// TIA Portal V20 export
DATA_BLOCK "DB_BadPartOnFixture"   // DB1308
{ S7_Optimized_Access := 'TRUE' }
// stored: AutoNumber false, MemoryReserve 100
   VAR
      BadPartOnFixture : Bool;
      ID_MeasureBad : Int;
   END_VAR
BEGIN
END_DATA_BLOCK
